Fanuc KAREL source: kt00553.KL

-- PROVISIONAL review KL for V940-1; original PC SHA256 09573262d87e722f603a7affb3d668fd4a6c071dfc72465c638a002cc2655f7c
-- Incomplete behavior may be omitted. Consult companion uncertainty JSON. Do not deploy.
PROGRAM KT00553
%NOLOCKGROUP
-- UNRESOLVED_DECL V1 type=000013
-- UNRESOLVED_DECL V2 type=000013
-- UNRESOLVED_DECL OUT type=000013
BEGIN
  -- V9_ZERO_TABLE_METADATA_HINT layout=0001; no indexed target words; source/name/runtime held
  -- UNRESOLVED_PC offsets 5-20; opcodes 2E,22,32,35
  -- UNRESOLVED_PC offsets 25-40; opcodes 2E,22,32,35
  -- UNRESOLVED_PC offsets 45-60; opcodes 2E,22,32,35
  -- UNRESOLVED_PC offsets 65-80; opcodes 2E,22,32,35
  -- UNRESOLVED_PC offsets 85-109; opcodes 49,49,91,4A
  -- UNRESOLVED_PC offsets 114-118; opcodes 7F
END KT00553
